// TIA Portal V19 export
TYPE "Prod_CIn"
   STRUCT
      Rst { ExternalWritable := 'False'} : Bool;
      Part_Execution { ExternalWritable := 'False'} : "Prod_Part_Done";
      Part_Prod { ExternalWritable := 'False'} : "Prod_Part_Area";
      Beam_Prod { ExternalWritable := 'False'} : "Prod_Beam_Area";
      Coil_Prod { ExternalWritable := 'False'} : "Prod_Coil_Area";
   END_STRUCT;
END_TYPE
